TYPE TFAxManCmd :
STRUCT
	
	Home	: BOOL	:= FALSE;	(* Home (Ricerca Posizione di Home) *)
	JogPos	: BOOL	:= FALSE;	(* Jog + *)
	JogNeg	: BOOL	:= FALSE;	(* Jog - *)
	JogFast	: BOOL	:= FALSE;	(* Jog +/- in Fast Speed *)
	
END_STRUCT
END_TYPE

(* stored: Version 1.1.0.1, ProductVersion 3.1.4024.11
   DUT TFAxManCmd: Id {aaa1fdc2-c972-4c26-b7fb-f00af5ff20b9} *)
